TYPE E_HmiCommandCode : (
    HMI_CMD_NONE := 0,
    HMI_CMD_START := 10,
    HMI_CMD_STOP := 20,
    HMI_CMD_INITIALIZE := 30,
    HMI_CMD_RESET := 40,
    HMI_CMD_ACK_RESULT := 50,
    HMI_CMD_SELECT_MAINTENANCE := 60,
    HMI_CMD_EXECUTE_MAINTENANCE := 70,
    HMI_CMD_CANCEL_MAINTENANCE := 80,
    HMI_CMD_VALIDATE_STEP := 90,
    HMI_CMD_SAVE_STEP := 100,
    HMI_CMD_VALIDATE_PROGRAM := 110,
    HMI_CMD_SAVE_PROGRAM := 120,
    HMI_CMD_ACTIVATE_PROGRAM := 130,
    HMI_CMD_SAVE_JOINING_POINT := 140,
    HMI_CMD_REQUEST_ALARM_PAGE := 150,
    HMI_CMD_REQUEST_CURVE_PAGE := 160
); END_TYPE

(* stored: Version 1.1.0.1
   DUT E_HmiCommandCode: Id {E3000000-0000-4000-8000-000000000023} *)
